% RSLogix 500 project P9 - DDE Messaging.RSS, saved by version 8.30.00.16 %
PROJECT "P9"    % processor: Bul.1763 MicroLogix 1100 Series B %

PROGRAM FILES
  LAD 2   10 rungs

DATA FILES
  O0 OUTPUT  4 elements
  I1 INPUT  6 elements
  S2 STATUS  66 elements
  B3 BINARY  1 elements
  T4 TIMER  4 elements
  C5 COUNTER  1 elements
  R6 CONTROL  1 elements
  N7 INTEGER  4 elements
  F8 FLOAT  1 elements
  ST9 STRING  8 elements

LADDER 2
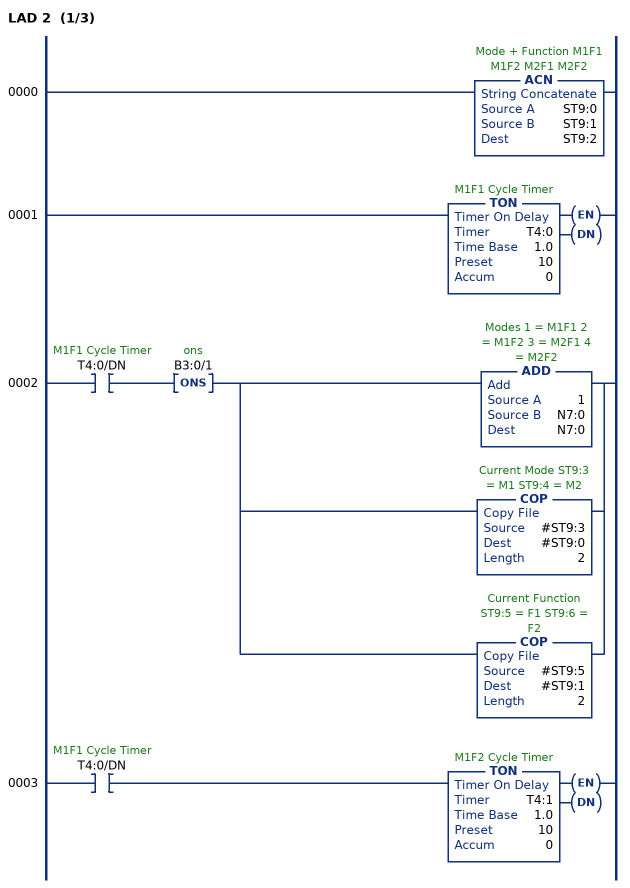
% Rung: 0 %
SOR ACN ST9:0 ST9:1 ST9:2 EOR
%   ST9:0  "Current Mode ST9:3 = M1 ST9:4 = M2" %
%   ST9:1  "Current Function ST9:5 = F1 ST9:6 = F2" %
%   ST9:2  "Mode + Function M1F1 M1F2 M2F1 M2F2" %
% Rung: 1 %
SOR TON T4:0 1.0 10 0 EOR
%   T4:0  "M1F1 Cycle Timer" %
% Rung: 2 %
SOR XIC T4:0/DN ONS B3:0/1 BST ADD 1 N7:0 N7:0 NXB COP #ST9:3 #ST9:0 2 NXB COP #ST9:5 #ST9:1 2 BND EOR
%   T4:0  "M1F1 Cycle Timer" %
%   B3:0/1  "ons" %
%   N7:0  "Modes 1 = M1F1 2 = M1F2 3 = M2F1 4 = M2F2" %
%   ST9:3  "String Search" %
%   ST9:0  "Current Mode ST9:3 = M1 ST9:4 = M2" %
%   ST9:5  "F1" %
%   ST9:1  "Current Function ST9:5 = F1 ST9:6 = F2" %
% Rung: 3 %
SOR XIC T4:0/DN TON T4:1 1.0 10 0 EOR
%   T4:0  "M1F1 Cycle Timer" %
%   T4:1  "M1F2 Cycle Timer" %

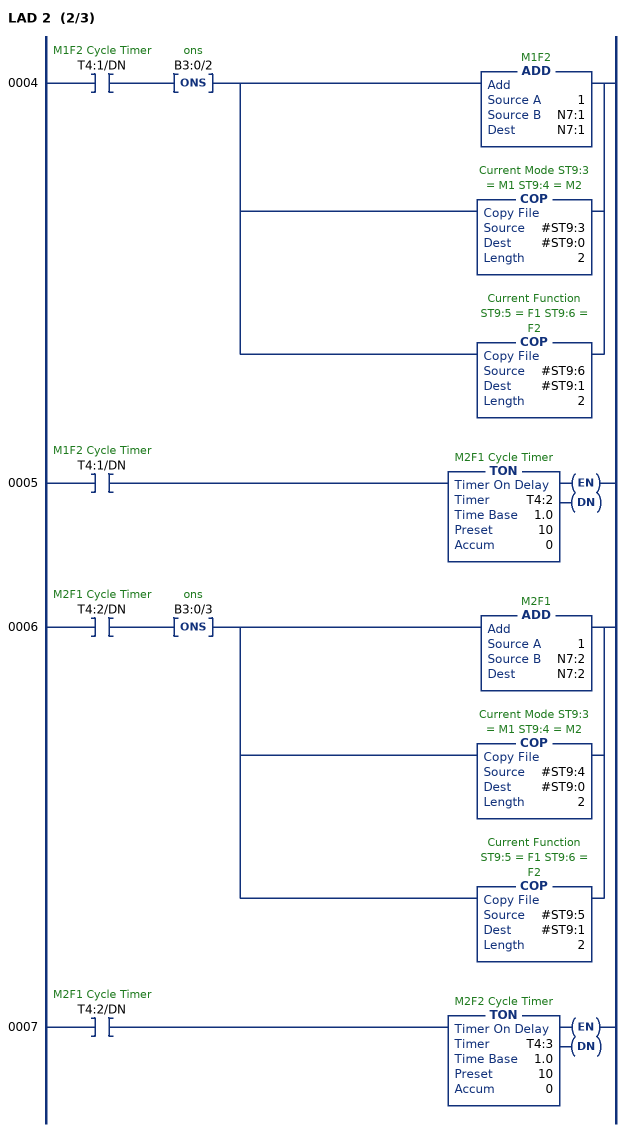
% Rung: 4 %
SOR XIC T4:1/DN ONS B3:0/2 BST ADD 1 N7:1 N7:1 NXB COP #ST9:3 #ST9:0 2 NXB COP #ST9:6 #ST9:1 2 BND EOR
%   T4:1  "M1F2 Cycle Timer" %
%   B3:0/2  "ons" %
%   N7:1  "M1F2" %
%   ST9:3  "String Search" %
%   ST9:0  "Current Mode ST9:3 = M1 ST9:4 = M2" %
%   ST9:6  "F2" %
%   ST9:1  "Current Function ST9:5 = F1 ST9:6 = F2" %
% Rung: 5 %
SOR XIC T4:1/DN TON T4:2 1.0 10 0 EOR
%   T4:1  "M1F2 Cycle Timer" %
%   T4:2  "M2F1 Cycle Timer" %
% Rung: 6 %
SOR XIC T4:2/DN ONS B3:0/3 BST ADD 1 N7:2 N7:2 NXB COP #ST9:4 #ST9:0 2 NXB COP #ST9:5 #ST9:1 2 BND EOR
%   T4:2  "M2F1 Cycle Timer" %
%   B3:0/3  "ons" %
%   N7:2  "M2F1" %
%   ST9:4  "M2" %
%   ST9:0  "Current Mode ST9:3 = M1 ST9:4 = M2" %
%   ST9:5  "F1" %
%   ST9:1  "Current Function ST9:5 = F1 ST9:6 = F2" %
% Rung: 7 %
SOR XIC T4:2/DN TON T4:3 1.0 10 0 EOR
%   T4:2  "M2F1 Cycle Timer" %
%   T4:3  "M2F2 Cycle Timer" %

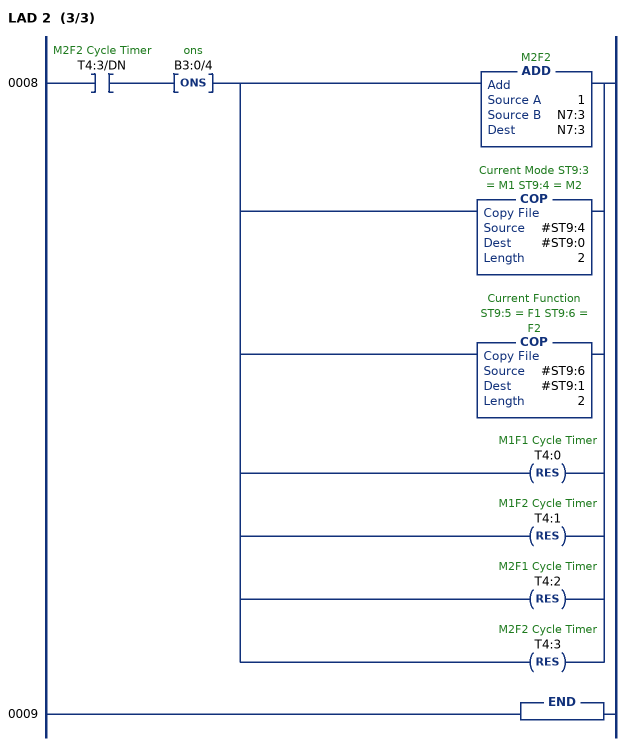
% Rung: 8 %
SOR XIC T4:3/DN ONS B3:0/4 BST ADD 1 N7:3 N7:3 NXB COP #ST9:4 #ST9:0 2 NXB COP #ST9:6 #ST9:1 2 NXB RES T4:0 NXB RES T4:1 NXB RES T4:2 NXB RES T4:3 BND EOR
%   T4:3  "M2F2 Cycle Timer" %
%   B3:0/4  "ons" %
%   N7:3  "M2F2" %
%   ST9:4  "M2" %
%   ST9:0  "Current Mode ST9:3 = M1 ST9:4 = M2" %
%   ST9:6  "F2" %
%   ST9:1  "Current Function ST9:5 = F1 ST9:6 = F2" %
%   T4:0  "M1F1 Cycle Timer" %
%   T4:1  "M1F2 Cycle Timer" %
%   T4:2  "M2F1 Cycle Timer" %
% Rung: 9 %
SOR END EOR

OTHER DOCUMENTED ADDRESSES
  B3:0/0  "Start Bit"
  B3:0/5  "Cycle Starter"
  C5:0  "M1F1 Counter"
  ST9:0.0  M1F1

DATA TABLE (non-zero values as saved)
DATA T4
% .PRE .ACC %
% T4:0 % 10 0
% T4:1 % 10 0
% T4:2 % 10 0
% T4:3 % 10 0
DATA ST9
% ST9:3 % "M1"
% ST9:4 % "M2"
% ST9:5 % "F1"
% ST9:6 % "F2"
